// TIA Portal V19 export
FUNCTION_BLOCK "BoilerAlarm"   // FB2, LAD
TITLE = Example of a Typed library block
{ S7_Optimized_Access := 'TRUE' }
// stored: MemoryReserve 100, SetENOAutomatically false
   VAR_INPUT
      "Alarm Bit" : Bool;
   END_VAR
   VAR
      Boiler : Program_Alarm;
   END_VAR
   VAR_TEMP
      "Return" : Int;
      "Current Time" : DTL;
      Boiler_Error : Bool;
      Boiler_Status : Word;
   END_VAR
BEGIN

REGION Network 1
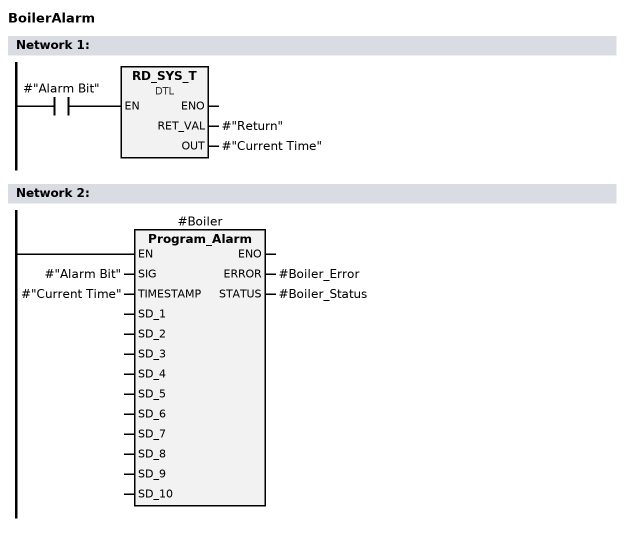
   RUNG wire#powerrail
      Contact( #"Alarm Bit" )
      { S7_Templates := "date_type := DTL" } RD_SYS_T(RET_VAL => #"Return", OUT => #"Current Time")
   END_RUNG
   // the same network as SCL:
   IF #"Alarm Bit" THEN #"Return" := RD_SYS_T(OUT => #"Current Time"); END_IF;
END_REGION

REGION Network 2
   RUNG wire#powerrail
      #Boiler.Program_Alarm(SIG := #"Alarm Bit", TIMESTAMP := #"Current Time", SD_1 :=, SD_2 :=, SD_3 :=, SD_4 :=, SD_5 :=, SD_6 :=, SD_7 :=, SD_8 :=, SD_9 :=, SD_10 :=, Error => #Boiler_Error, Status => #Boiler_Status)
   END_RUNG
   // the same network as SCL:
   #Boiler(SIG := #"Alarm Bit", TIMESTAMP := #"Current Time", Error => #Boiler_Error, Status => #Boiler_Status);   // Program_Alarm
END_REGION
END_FUNCTION_BLOCK
